FUNCTION_BLOCK FB_MachineInfo
VAR_INPUT 
	Trigger				: BOOL;
	RemoveRouteName		: STRING;
	RemoveRoute			: BOOL;
END_VAR
VAR_OUTPUT
	Adapters 			: ARRAY[0..MAX_LOCAL_ADAPTERS] OF ST_IpAdapterInfo;
	Licenses   			: ARRAY[1..nMaxLicenses] OF ST_TcOnlineLicenseInfoData;
	Routes				: ARRAY[0..15] OF ST_AmsRouteEntry;
END_VAR
VAR PERSISTENT
	NetworkDevices 		: ARRAY[0..15] OF ST_IpAdapterInfo;
END_VAR

M_CPU();

METHOD M_CPU
VAR_STAT
	_GetAdaptersInfo	: FB_GetAdaptersInfo;
	_GetLicenses		: FB_GetLicenses;
	_EnumRouteEntry		: FB_EnumRouteEntry;
	_RemoveRouteEntry 	: FB_RemoveRouteEntry;
	_incrementer		: INT;
	_x					: INT;
	_y					: INT;
	_step				: INT;
END_VAR
CASE _step OF
	0 :
		_GetAdaptersInfo.bExecute := FALSE;
		_GetLicenses.bExecute := FALSE;
		_EnumRouteEntry.bExecute := FALSE;
		_EnumRouteEntry.eCmd := eEnumCmd_First;
		_RemoveRouteEntry.bExecute := FALSE;
		_incrementer:=0;
		Trigger:=FALSE;
		_step:=_step+1;

	1 :
		_EnumRouteEntry.bExecute := TRUE;
		IF _EnumRouteEntry.bBusy THEN
		_step:=_step+1; END_IF
	
	2 :
		_EnumRouteEntry.bExecute := FALSE;
		IF NOT _EnumRouteEntry.bBusy THEN
		_step:=_step+1; END_IF
	
	3 :
		IF _EnumRouteEntry.bEOE THEN
			_step:=_step+1; 
			FOR _incrementer := _incrementer TO 15 BY 1 DO
				Routes[_incrementer].dwFlags:=0;
				Routes[_incrementer].eTransport:=0;
				Routes[_incrementer].sAddress:='';
				Routes[_incrementer].sName:='';
				Routes[_incrementer].sNetID:='';
				Routes[_incrementer].tTimeout:=T#0S;
			END_FOR
		ELSE
			Routes[_incrementer]:= _EnumRouteEntry.stRoute;
			_incrementer := _incrementer + 1;
			_EnumRouteEntry.eCmd := eEnumCmd_Next;
			_step:=1;
		END_IF
		
	4 :
		_GetAdaptersInfo.bExecute := TRUE;
		IF _GetAdaptersInfo.bBusy THEN
		_step:=_step+1; END_IF
			
	5 :
		_GetAdaptersInfo.bExecute := FALSE;
		IF NOT _GetAdaptersInfo.bBusy THEN
		_step:=_step+1; END_IF
				
	6 :
		_GetLicenses.bExecute := TRUE;
		IF _GetLicenses.bBusy THEN
		_step:=_step+1; END_IF
				
	7 :
		_GetLicenses.bExecute := FALSE;
		IF NOT _GetLicenses.bBusy THEN
		_step:=_step+1; END_IF
		
	8 :
		Adapters := _GetAdaptersInfo.arrAdapters;
		IF _GetLicenses.nValidLicenses > 0 THEN
			FOR _incrementer := 1 TO UDINT_TO_INT(_GetLicenses.nValidLicenses) DO
				Licenses[_incrementer] := _GetLicenses.aValidLicenses[_incrementer];
			END_FOR
		END_IF
		IF _GetLicenses.nInvalidLicenses > 0 THEN
			FOR _incrementer := UDINT_TO_INT(_GetLicenses.nValidLicenses+1) TO UDINT_TO_INT(_GetLicenses.nValidLicenses + _GetLicenses.nInvalidLicenses) DO
				Licenses[_incrementer] := _GetLicenses.aInvalidLicenses[_incrementer-UDINT_TO_INT(_GetLicenses.nInvalidLicenses)];
			END_FOR
		END_IF
		_step:=_step+1;
		
	9 :
		IF Trigger THEN _step:=0; END_IF
		IF RemoveRoute THEN _step:=_step+1; END_IF
		
	10:
		_RemoveRouteEntry.sName := RemoveRouteName;
		_RemoveRouteEntry.bExecute := TRUE;
		IF _RemoveRouteEntry.bBusy THEN
		_step:=_step+1; END_IF
			
	11:
		_RemoveRouteEntry.bExecute := FALSE;
		IF NOT _RemoveRouteEntry.bBusy THEN
		RemoveRoute := FALSE;
		_step:=0; END_IF
		
ELSE
	_step:=0;
END_CASE

_GetAdaptersInfo();
_GetLicenses();
_EnumRouteEntry();
_RemoveRouteEntry();
END_METHOD

END_FUNCTION_BLOCK

(* stored: Version 1.1.0.1, ProductVersion 3.1.4024.3
   POU FB_MachineInfo: Id {378bffd0-be4c-44b9-af66-722f0b9499f2}, SpecialFunc None
   Method M_CPU: Id {a4f384af-9b7e-40c5-a9ac-7afcfe0bf912} *)
